# EPICS autosave request: calcApp/Db/userAve_settings.req
$(P)userAve$(N).DESC
$(P)userAve$(N).SCAN
$(P)userAve$(N).INPB
$(P)userAve$(N).A
$(P)userAve$(N).PREC
$(P)userAve$(N)_mode
$(P)userAve$(N)_algorithm
$(P)userAve$(N).FLNK
